// TIA Portal project "Automatic_Welder_1.0.0" (V19)
// Separate project file needed for simulation as  It was never possible to simulate an S7-1200 with firmware V3.0. It became only available with the firmware V4.0. Before this we had to use an S7-1500 to simulate the process.
// 
// The physical CPU cannot upgrade to firmware V3.0 -> V4.0. But software allows changing a V3.0 with V4.0 CPU. Downgrading a V4.0 project to V3.0 is not directly possible and is very painful.
// 
// The very best is to have two PLC projects. One is the design version (V3.0) and the other the simulation version (V4.0). Copy changes over from one to the other as needed.
// 
// The next option is to have a physical PLC at your desk. Ask your supplier to lend you a demo module from an old demo kit.

(* hardware
DEVICE "HMI_1"  TP700 Comfort
   slot 0: "HMI_1"  TP700 Comfort  6AV2 124-0GC01-0AX0  17.0.0.0
   slot 1: "HMI_1"  TP700 Comfort  6AV2 124-0GC01-0AX0  17.0.0.0
   slot 5: "HMI_1.IE_CP_1"  PROFINET Interface  17.0.0.0
      slot 1: "PROFINET Interface_1"  PROFINET Interface
         slot 1: "Port_1"  Port
         slot 2: "Port_2"  Port
   slot 7: "HMI_1.MPI/DP_CP_1"  MPI/DP Interface  17.0.0.0
DEVICE "S7-1200 station_1"  S7-1200 Station
   slot 0: "Rack_0"  S7-1200 Rack  Rack  V1.0
   slot 1: "PLC_1"  CPU 1214C DC/DC/DC  6ES7 214-1AG40-0XB0  V4.6
*)

// ===== PLC "PLC_1"  CPU 1214C DC/DC/DC =====

VAR_GLOBAL   // PLC tag table "Program Control"
   "ProgramStarted" AT %M0.1 : Bool;   // change to I instead of M later on
   "ProgramPaused" AT %M0.2 : Bool;   // change to I instead of M later on
   "SentCommandMoveXY" AT %M0.3 : Bool;   // being buggy and weird
   "SystemStatus" AT %QW1 : Int;   // codes: 100 - ok. 201 - motor address error
   "EnableMotorXY" AT %M0.0 : Bool;
END_VAR

VAR_GLOBAL   // PLC tag table "Clock_Memory"
   "Clock_Byte" AT %MB100 : Byte;
   "Clock_10Hz" AT %M100.0 : Bool;
   "Clock_5Hz" AT %M100.1 : Bool;
   "Clock_2.5Hz" AT %M100.2 : Bool;
   "Clock_2Hz" AT %M100.3 : Bool;
   "Clock_1.25Hz" AT %M100.4 : Bool;
   "Clock_1Hz" AT %M100.5 : Bool;
   "Clock_0.625Hz" AT %M100.6 : Bool;
   "Clock_0.5Hz" AT %M100.7 : Bool;
END_VAR

DATA_BLOCK "User_IO_DB"   // DB1
{ S7_Optimized_Access := 'TRUE' }
VERSION : 0.1
   VAR
      XSpeed : UDInt := 0;   // Pulse /hz
      XDest : UDInt;
      XPulses : DInt := 0;   // 21800 Pulse / 2mm
      XValue : UDInt := 0;   // 384-16=368u
      YSpeed : UDInt := 0;   // Pulse /hz
      YPulses : DInt := 0;   // 21800 Pulse / 2mm
      YDest : UDInt;
      Yvalue : UDInt := 0;   // 456-152=304u
   END_VAR
BEGIN
END_DATA_BLOCK

DATA_BLOCK "System_Update_DB"   // DB2
{ S7_Optimized_Access := 'TRUE' }
VERSION : 0.1
   VAR
      EnableMotorXYB : Bool;
      RunTerminationDone : Bool;
      RunStartupDone : Bool;
      DoneMotorX : Bool;
      DoneMotorXB : Bool;
      DoneMotorY : Bool;
      DoneMotorYB : Bool;
   END_VAR
BEGIN
END_DATA_BLOCK

DATA_BLOCK "Test_DB"   // DB3
{ S7_Optimized_Access := 'TRUE' }
VERSION : 0.1
   VAR
      "a" : DInt;
      aa : DInt;
      aaa : UDInt;
      aaaa : UDInt;
      "b" : Bool;
      bb : Bool;
      bbb : Bool;
      c : Time;
      dd : Real;
      d : Real;
      bbbb : Bool;
   END_VAR
BEGIN
END_DATA_BLOCK

// folder: Stepper Motor

DATA_BLOCK "X_Motor_Feedback_DB"   // DB5
{ S7_Optimized_Access := 'TRUE' }
VERSION : 0.1
// stored: InstanceOfName Motor_Feedback
"Motor_Feedback"
BEGIN
END_DATA_BLOCK

DATA_BLOCK "Y_Motor_Feedback_DB"   // DB6
{ S7_Optimized_Access := 'TRUE' }
VERSION : 0.1
// stored: InstanceOfName Motor_Feedback
"Motor_Feedback"
BEGIN
END_DATA_BLOCK

// folder: System blocks/Program resources

DATA_BLOCK "Motor_TimesUp_DB"   // DB4
{ S7_Optimized_Access := 'TRUE' }
AUTHOR : Simatic
FAMILY : IEC
NAME : IEC_TMR
VERSION : 1.0
// stored: InstanceOfName IEC_TIMER
"IEC_TIMER"
BEGIN
END_DATA_BLOCK

// folder: (top level)

ORGANIZATION_BLOCK "Main"   // OB1, LAD, ProgramCycle
TITLE = "Main Program Sweep (Cycle)"
{ S7_Optimized_Access := 'TRUE' }
VERSION : 0.1
   VAR_INPUT
      Initial_Call : Bool;   // Initial call of this OB
      Remanence : Bool;   // =True, if remanent data are available
   END_VAR
   VAR_TEMP
      XSucceeded : Bool;
      YSucceeded : Bool;
      Tmp : Bool;
      Tmp2 : Bool;
      TmpB : Bool;
   END_VAR
   VAR_TEMP   // added for the SCL form of the ladder/FBD networks
      _w1 : Bool;
      _w2 : Bool;
      _w3 : Bool;
      _w4 : Bool;
   END_VAR
BEGIN

REGION Network 1: Handle Motor UserInput
   // todo: need to size conversion for pulses, distance (mm), hmi distance (a.u.), del ismoving (redundant)
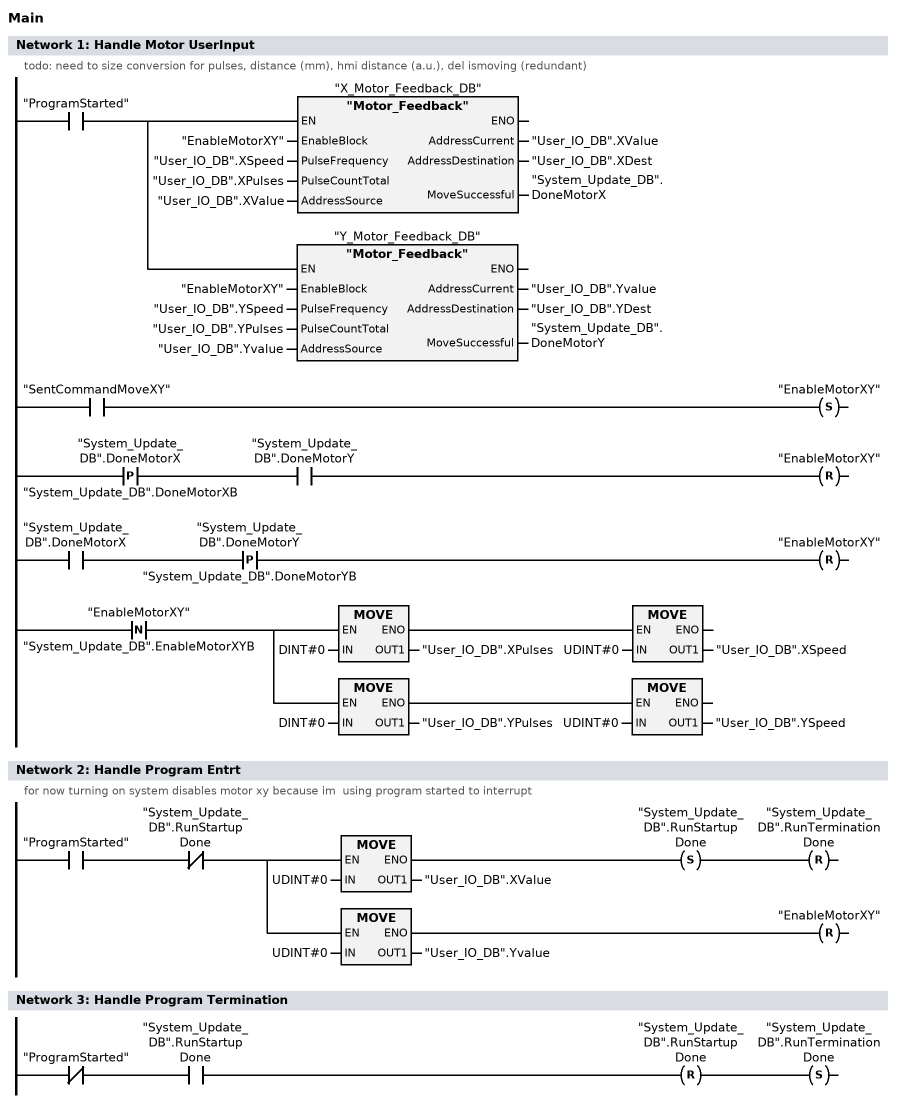
   RUNG wire#powerrail
      Contact( "ProgramStarted" )
      wire#w1
      "X_Motor_Feedback_DB"(EnableBlock := "EnableMotorXY", PulseFrequency := "User_IO_DB".XSpeed, PulseCountTotal := "User_IO_DB".XPulses, AddressSource := "User_IO_DB".XValue, AddressCurrent => "User_IO_DB".XValue, AddressDestination => "User_IO_DB".XDest, MoveSuccessful => "System_Update_DB".DoneMotorX)
   END_RUNG
   RUNG wire#w1
      "Y_Motor_Feedback_DB"(EnableBlock := "EnableMotorXY", PulseFrequency := "User_IO_DB".YSpeed, PulseCountTotal := "User_IO_DB".YPulses, AddressSource := "User_IO_DB".Yvalue, AddressCurrent => "User_IO_DB".Yvalue, AddressDestination => "User_IO_DB".YDest, MoveSuccessful => "System_Update_DB".DoneMotorY)
   END_RUNG
   RUNG wire#powerrail
      Contact( "SentCommandMoveXY" )
      S_Coil( "EnableMotorXY" )
   END_RUNG
   RUNG wire#powerrail
      P_Contact(operand := "System_Update_DB".DoneMotorX, bit := "System_Update_DB".DoneMotorXB)
      Contact( "System_Update_DB".DoneMotorY )
      R_Coil( "EnableMotorXY" )
   END_RUNG
   RUNG wire#powerrail
      Contact( "System_Update_DB".DoneMotorX )
      P_Contact(operand := "System_Update_DB".DoneMotorY, bit := "System_Update_DB".DoneMotorYB)
      R_Coil( "EnableMotorXY" )
   END_RUNG
   RUNG wire#powerrail
      N_Contact(operand := "EnableMotorXY", bit := "System_Update_DB".EnableMotorXYB)
      wire#w2
      Move(in := DINT#0, out1 => "User_IO_DB".XPulses)
      Move(in := UDINT#0, out1 => "User_IO_DB".XSpeed)
   END_RUNG
   RUNG wire#w2
      Move(in := DINT#0, out1 => "User_IO_DB".YPulses)
      Move(in := UDINT#0, out1 => "User_IO_DB".YSpeed)
   END_RUNG
   // the same network as SCL:
   #_w1 := "ProgramStarted";
   IF #_w1 THEN
       "X_Motor_Feedback_DB"(EnableBlock := "EnableMotorXY",   // "Motor_Feedback"
                             PulseFrequency := "User_IO_DB".XSpeed,
                             PulseCountTotal := "User_IO_DB".XPulses,
                             AddressSource := "User_IO_DB".XValue,
                             AddressCurrent => "User_IO_DB".XValue,
                             AddressDestination => "User_IO_DB".XDest,
                             MoveSuccessful => "System_Update_DB".DoneMotorX);
       "Y_Motor_Feedback_DB"(EnableBlock := "EnableMotorXY",   // "Motor_Feedback"
                             PulseFrequency := "User_IO_DB".YSpeed,
                             PulseCountTotal := "User_IO_DB".YPulses,
                             AddressSource := "User_IO_DB".Yvalue,
                             AddressCurrent => "User_IO_DB".Yvalue,
                             AddressDestination => "User_IO_DB".YDest,
                             MoveSuccessful => "System_Update_DB".DoneMotorY);
   END_IF;
   IF "SentCommandMoveXY" THEN "EnableMotorXY" := TRUE; END_IF;
   #_w2 := "System_Update_DB".DoneMotorX AND NOT "System_Update_DB".DoneMotorXB;   // rising edge of "System_Update_DB".DoneMotorX
   "System_Update_DB".DoneMotorXB := "System_Update_DB".DoneMotorX;
   IF #_w2 AND "System_Update_DB".DoneMotorY THEN "EnableMotorXY" := FALSE; END_IF;
   #_w3 := "System_Update_DB".DoneMotorX AND "System_Update_DB".DoneMotorY AND NOT "System_Update_DB".DoneMotorYB;   // rising edge of "System_Update_DB".DoneMotorY
   "System_Update_DB".DoneMotorYB := "System_Update_DB".DoneMotorY;
   IF #_w3 THEN "EnableMotorXY" := FALSE; END_IF;
   #_w4 := NOT "EnableMotorXY" AND "System_Update_DB".EnableMotorXYB;   // falling edge of "EnableMotorXY"
   "System_Update_DB".EnableMotorXYB := "EnableMotorXY";
   IF #_w4 THEN
       "User_IO_DB".XPulses := DINT#0;
       "User_IO_DB".XSpeed := UDINT#0;
       "User_IO_DB".YPulses := DINT#0;
       "User_IO_DB".YSpeed := UDINT#0;
   END_IF;
END_REGION

REGION Network 2: Handle Program Entrt
   // for now turning on system disables motor xy because im  using program started to interrupt
   RUNG wire#powerrail
      Contact( "ProgramStarted" )
      I_Contact( "System_Update_DB".RunStartupDone )
      wire#w1
      Move(in := UDINT#0, out1 => "User_IO_DB".XValue)
      S_Coil( "System_Update_DB".RunStartupDone )
      R_Coil( "System_Update_DB".RunTerminationDone )
   END_RUNG
   RUNG wire#w1
      Move(in := UDINT#0, out1 => "User_IO_DB".Yvalue)
      R_Coil( "EnableMotorXY" )
   END_RUNG
   // the same network as SCL:
   IF "ProgramStarted" AND NOT "System_Update_DB".RunStartupDone THEN "User_IO_DB".XValue := UDINT#0; END_IF;
   #_w1 := "ProgramStarted" AND NOT "System_Update_DB".RunStartupDone;
   IF #_w1 THEN
       "System_Update_DB".RunStartupDone := TRUE;
       "System_Update_DB".RunTerminationDone := FALSE;
       "User_IO_DB".Yvalue := UDINT#0;
       "EnableMotorXY" := FALSE;
   END_IF;
END_REGION

REGION Network 3: Handle Program Termination
   RUNG wire#powerrail
      I_Contact( "ProgramStarted" )
      Contact( "System_Update_DB".RunStartupDone )
      R_Coil( "System_Update_DB".RunStartupDone )
      S_Coil( "System_Update_DB".RunTerminationDone )
   END_RUNG
   // the same network as SCL:
   #_w1 := NOT "ProgramStarted" AND "System_Update_DB".RunStartupDone;
   IF #_w1 THEN
       "System_Update_DB".RunStartupDone := FALSE;
       "System_Update_DB".RunTerminationDone := TRUE;
   END_IF;
END_REGION
END_ORGANIZATION_BLOCK

ORGANIZATION_BLOCK "Test_CyclicOB"   // OB123, LAD, ProgramCycle
TITLE = "Main Program Sweep (Cycle)"
{ S7_Optimized_Access := 'TRUE' }
VERSION : 0.1
   VAR_INPUT
      Initial_Call : Bool;   // Initial call of this OB
      Remanence : Bool;   // =True, if remanent data are available
   END_VAR
   VAR_TEMP
      tb : Bool;
      tbb : Bool;
      var_time1 : Real;
      var_time2 : UDInt;
      tbEdgeDetected : Bool;
   END_VAR
   VAR_TEMP   // added for the SCL form of the ladder/FBD networks
      _w1 : Bool;
   END_VAR
BEGIN

REGION Network 1: Ladder logic (I am retarded)
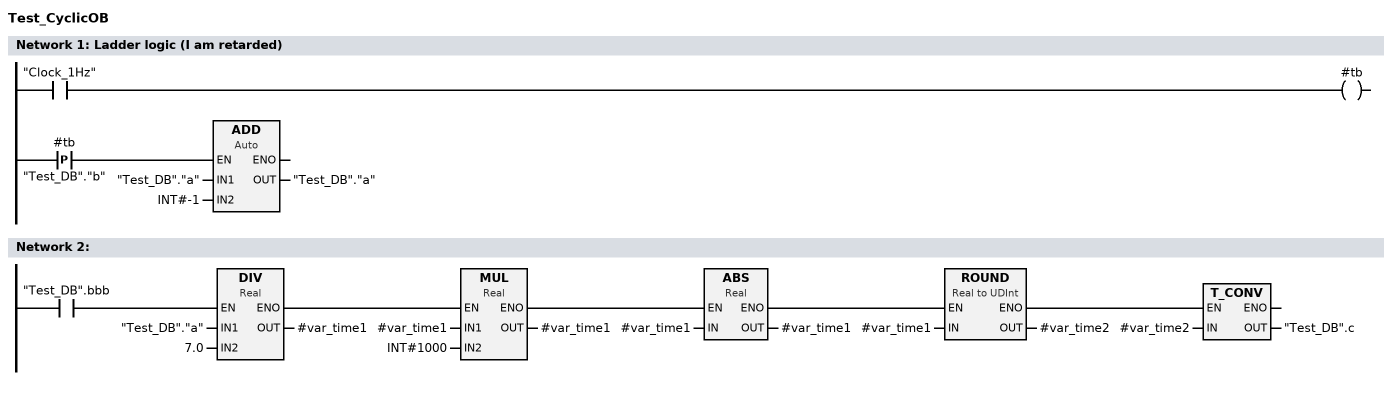
   RUNG wire#powerrail
      Contact( "Clock_1Hz" )
      Coil( #tb )
   END_RUNG
   RUNG wire#powerrail
      P_Contact(operand := #tb, bit := "Test_DB"."b")
      Add(in1 := "Test_DB"."a", in2 := INT#-1, out => "Test_DB"."a")
   END_RUNG
   // the same network as SCL:
   #tb := "Clock_1Hz";
   #_w1 := #tb AND NOT "Test_DB"."b";   // rising edge of #tb
   "Test_DB"."b" := #tb;
   IF #_w1 THEN "Test_DB"."a" := "Test_DB"."a" + INT#-1; END_IF;
END_REGION

REGION Network 2
   IF "Test_DB".bbb THEN
       #var_time1 := "Test_DB"."a" / 7.0;
       #var_time1 := #var_time1 * INT#1000;
       #var_time1 := ABS(#var_time1);
       #var_time2 := ROUND(#var_time1);
       "Test_DB".c := T_CONV(IN := #var_time2);
   END_IF;
END_REGION

REGION Network 3 (SCL): turn pulses into time (ms)
   #var_time1 := "Test_DB".a / 7;
   #var_time1 := ABS(#var_time1 * 1000);
   #var_time2 := REAL_TO_UDINT(#var_time1);
   "Test_DB".c := UDINT_TO_TIME(#var_time2);
END_REGION
END_ORGANIZATION_BLOCK

// folder: Stepper Motor

FUNCTION_BLOCK "Motor_Feedback"   // FB2, LAD
TITLE = Motor Telemetry: Get current axis position and if the motor is moving.
{ S7_Optimized_Access := 'TRUE' }
VERSION : 0.1
// TODO: Make block figure out when to allow the motor to stop moving (So that the current location is known.) when a move operation is interrupted.
// Implement reversed movement logic
// 
// Motor movement logic is currently only in blocks of pulse per 500ms except for final, ratify this.
// go test if can change the static vars to temp
// 
// d = vt
// pulses = pulsefrequency times time
// go figure out how far one pulse moves,  bi/unipolar, do conversions to metric!
   VAR_INPUT
      EnableBlock : Bool;
      PulseFrequency : DInt;   // hz
      PulseCountTotal : DInt;
      AddressSource : DInt;
   END_VAR
   VAR_OUTPUT
      AddressCurrent : DInt;
      AddressDestination : Int;
      MoveSuccessful : Bool;
   END_VAR
   VAR
      TimeTotalms : Time;
      PulseCountDone : DInt;
      Movement500ms : DInt;
      IsMoving : Bool;
      IsMovingM : Bool;
      TimerDiff : Bool;
      TimerDiffB : Bool;
      EnableBlockM : Bool;
   END_VAR
   VAR_TEMP
      IsPulseCountNegative : SInt;
      PulseCountAbs : UDInt;
   END_VAR
   VAR_TEMP   // added for the SCL form of the ladder/FBD networks
      _w1 : Bool;
      _w2 : Bool;
   END_VAR
BEGIN

REGION Network 1: ENTRY Evaluate Working Variables + Call Main
   // I spent 2 hours on this: Scan Op for positve edge can only be used for one row! This is because it ref the same bit.
   // 
   // Find:
   // - Move Destination
   // - Time total (ms): PulseCountTotal = PulseFrequency(hz) * Time (s)
   // - Pulses / 500ms (auto rounded by DIV)
   // - Current Address = Source Address
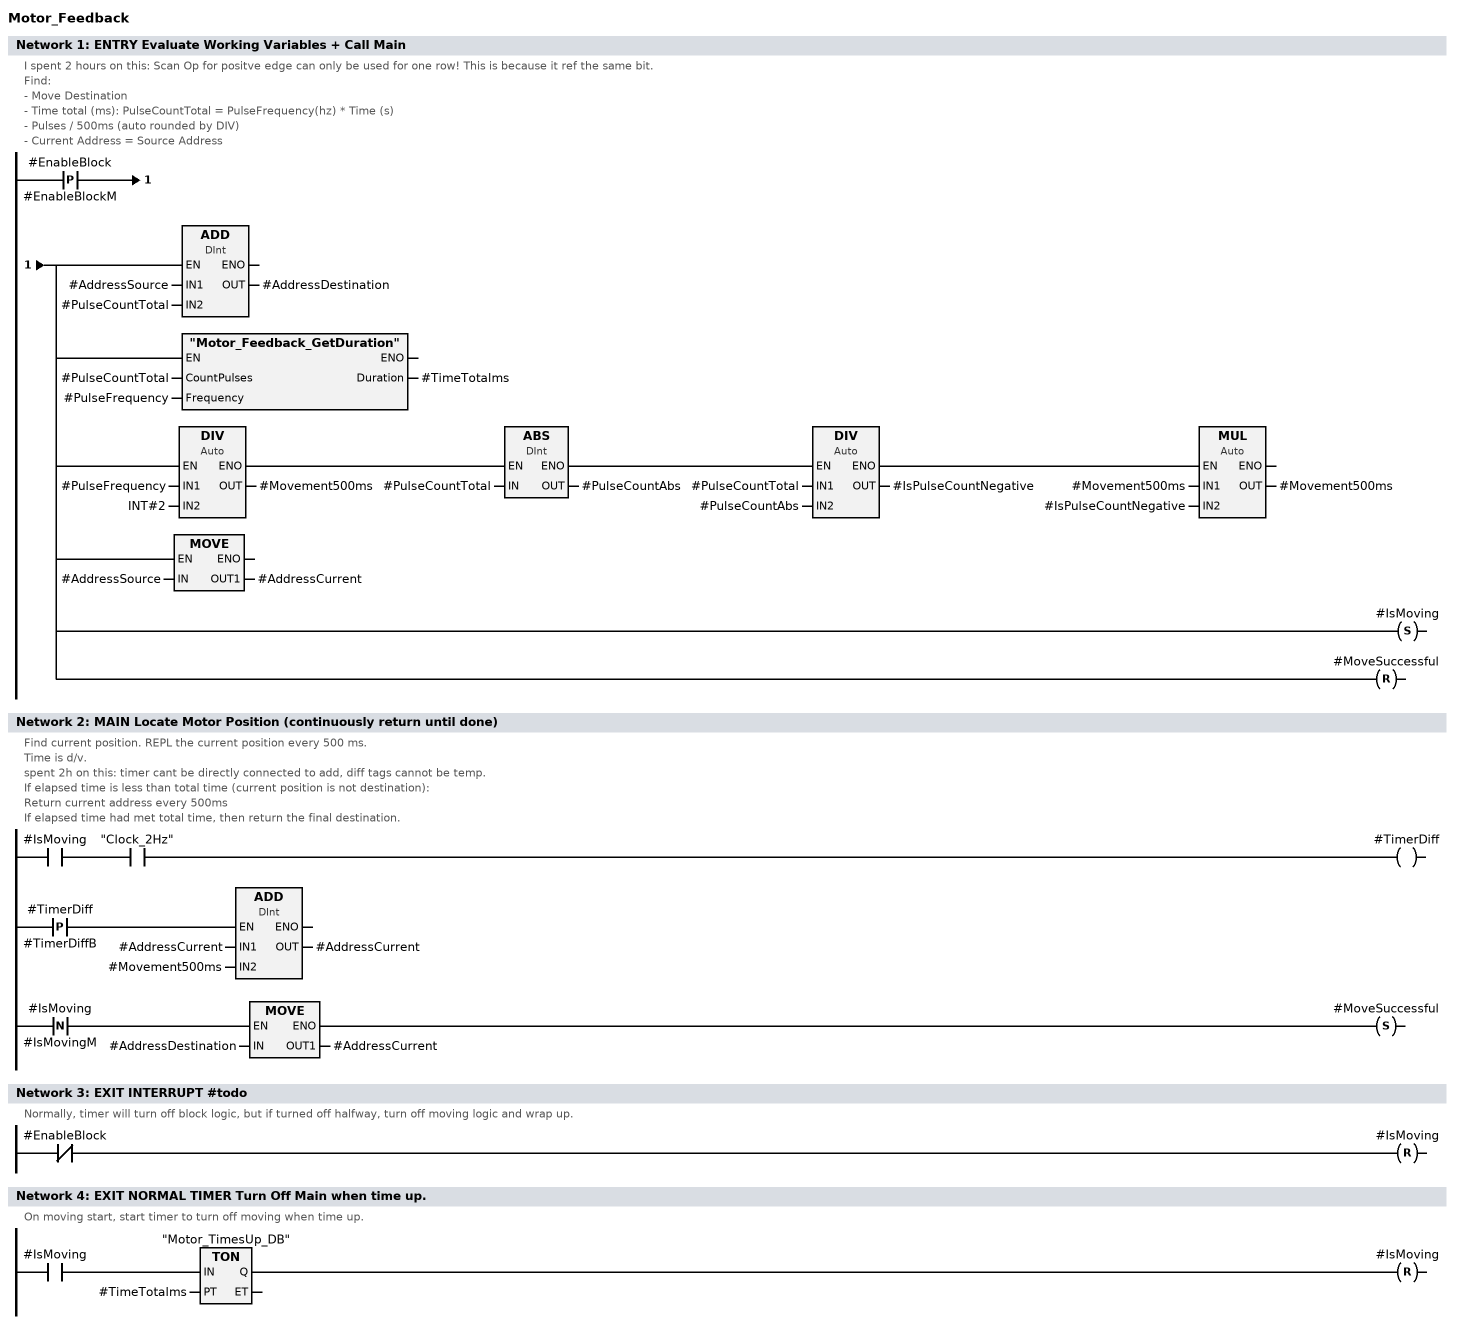
   RUNG wire#powerrail
      P_Contact(operand := #EnableBlock, bit := #EnableBlockM)
      wire#w1
      { S7_Templates := "SrcType := DInt" } Add(in1 := #AddressSource, in2 := #PulseCountTotal, out => #AddressDestination)
   END_RUNG
   RUNG wire#w1
      "Motor_Feedback_GetDuration"(CountPulses := #PulseCountTotal, Frequency := #PulseFrequency, Duration => #TimeTotalms)
   END_RUNG
   RUNG wire#w1
      Div(in1 := #PulseFrequency, in2 := INT#2, out => #Movement500ms)
      { S7_Templates := "SrcType := DInt" } Abs(in := #PulseCountTotal, out => #PulseCountAbs)
      Div(in1 := #PulseCountTotal, in2 := #PulseCountAbs, out => #IsPulseCountNegative)
      Mul(in1 := #Movement500ms, in2 := #IsPulseCountNegative, out => #Movement500ms)
   END_RUNG
   RUNG wire#w1
      Move(in := #AddressSource, out1 => #AddressCurrent)
   END_RUNG
   RUNG wire#w1
      S_Coil( #IsMoving )
   END_RUNG
   RUNG wire#w1
      R_Coil( #MoveSuccessful )
   END_RUNG
   // the same network as SCL:
   #_w1 := #EnableBlock AND NOT #EnableBlockM;   // rising edge of #EnableBlock
   #EnableBlockM := #EnableBlock;
   IF #_w1 THEN
       #AddressDestination := #AddressSource + #PulseCountTotal;
       "Motor_Feedback_GetDuration"(CountPulses := #PulseCountTotal,
                               Frequency := #PulseFrequency,
                               Duration => #TimeTotalms);
       #Movement500ms := #PulseFrequency / INT#2;
       #PulseCountAbs := ABS(#PulseCountTotal);
       #IsPulseCountNegative := #PulseCountTotal / #PulseCountAbs;
       #Movement500ms := #Movement500ms * #IsPulseCountNegative;
       #AddressCurrent := #AddressSource;
       #IsMoving := TRUE;
       #MoveSuccessful := FALSE;
   END_IF;
END_REGION

REGION Network 2: MAIN Locate Motor Position (continuously return until done)
   // Find current position. REPL the current position every 500 ms.
   // Time is d/v. 
   // 
   // spent 2h on this: timer cant be directly connected to add, diff tags cannot be temp.
   // 
   // If elapsed time is less than total time (current position is not destination):
   // Return current address every 500ms
   // 
   // If elapsed time had met total time, then return the final destination.
   RUNG wire#powerrail
      Contact( #IsMoving )
      Contact( "Clock_2Hz" )
      Coil( #TimerDiff )
   END_RUNG
   RUNG wire#powerrail
      P_Contact(operand := #TimerDiff, bit := #TimerDiffB)
      { S7_Templates := "SrcType := DInt" } Add(in1 := #AddressCurrent, in2 := #Movement500ms, out => #AddressCurrent)
   END_RUNG
   RUNG wire#powerrail
      N_Contact(operand := #IsMoving, bit := #IsMovingM)
      Move(in := #AddressDestination, out1 => #AddressCurrent)
      S_Coil( #MoveSuccessful )
   END_RUNG
   // the same network as SCL:
   #TimerDiff := #IsMoving AND "Clock_2Hz";
   #_w1 := #TimerDiff AND NOT #TimerDiffB;   // rising edge of #TimerDiff
   #TimerDiffB := #TimerDiff;
   IF #_w1 THEN #AddressCurrent := #AddressCurrent + #Movement500ms; END_IF;
   #_w2 := NOT #IsMoving AND #IsMovingM;   // falling edge of #IsMoving
   #IsMovingM := #IsMoving;
   IF #_w2 THEN
       #AddressCurrent := #AddressDestination;
       #MoveSuccessful := TRUE;
   END_IF;
END_REGION

REGION Network 3: EXIT INTERRUPT #todo
   // Normally, timer will turn off block logic, but if turned off halfway, turn off moving logic and wrap up.
   RUNG wire#powerrail
      I_Contact( #EnableBlock )
      R_Coil( #IsMoving )
   END_RUNG
   // the same network as SCL:
   IF NOT #EnableBlock THEN #IsMoving := FALSE; END_IF;
END_REGION

REGION Network 4: EXIT NORMAL TIMER Turn Off Main when time up.
   // On moving start, start timer to turn off moving when time up.
   "Motor_TimesUp_DB".TON(IN := #IsMoving, PT := #TimeTotalms);
   IF "Motor_TimesUp_DB".Q THEN #IsMoving := FALSE; END_IF;
END_REGION
END_FUNCTION_BLOCK

FUNCTION_BLOCK "Motor_Commands"   // FB3, LAD
{ S7_Optimized_Access := 'TRUE' }
VERSION : 0.1
   VAR_OUTPUT
      Pulse : Bool;
   END_VAR
BEGIN
END_FUNCTION_BLOCK

FUNCTION "Motor_Feedback_GetDuration" : Void   // FC1, SCL
{ S7_Optimized_Access := 'TRUE' }
VERSION : 0.1
   VAR_INPUT
      CountPulses : DInt;
      Frequency : DInt;
   END_VAR
   VAR_OUTPUT
      Duration : Time;
   END_VAR
   VAR_TEMP
      x0 : Real;
      x1 : UDInt;
   END_VAR
BEGIN
   #x0 := #CountPulses / #Frequency; // real output
   #x0 := ABS(#x0 * 1000);
   #x1 := REAL_TO_UDINT(#x0);
   #Duration := UDINT_TO_TIME(#x1);
END_FUNCTION

FUNCTION "Motor_Feedback_GetMovement" : Void   // FC2, LAD
{ S7_Optimized_Access := 'TRUE' }
VERSION : 0.1
   VAR_INPUT
      PulseFrequency : UDInt;
      PulseCount : DInt;
      ClockInterval : USInt;
   END_VAR
   VAR_OUTPUT
      MovementUnit : DInt;
   END_VAR
   VAR_TEMP
      PulseCountAbs : UDInt;
      IsPulseCountNegative : SInt;
      MovementUnitAbs : UDInt;
   END_VAR
BEGIN

REGION Network 1
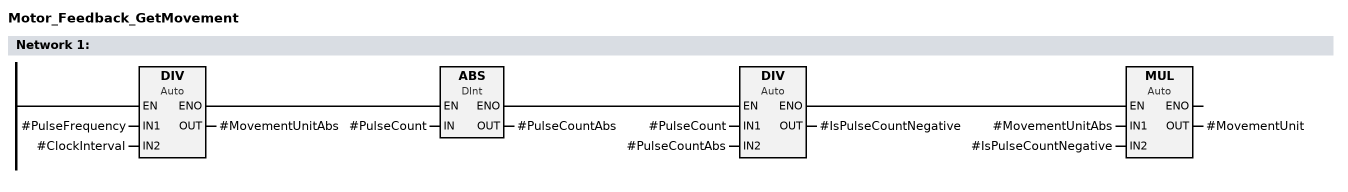
   RUNG wire#powerrail
      Div(in1 := #PulseFrequency, in2 := #ClockInterval, out => #MovementUnitAbs)
      { S7_Templates := "SrcType := DInt" } Abs(in := #PulseCount, out => #PulseCountAbs)
      Div(in1 := #PulseCount, in2 := #PulseCountAbs, out => #IsPulseCountNegative)
      Mul(in1 := #MovementUnitAbs, in2 := #IsPulseCountNegative, out => #MovementUnit)
   END_RUNG
   // the same network as SCL:
   #MovementUnitAbs := #PulseFrequency / #ClockInterval;
   #PulseCountAbs := ABS(#PulseCount);
   #IsPulseCountNegative := #PulseCount / #PulseCountAbs;
   #MovementUnit := #MovementUnitAbs * #IsPulseCountNegative;
END_REGION
END_FUNCTION

(* ===== HMI "HMI_1" =====
system functions are stored by id; their names below are inferred from use
connection "HMI_Connection_2": ETHERNET, S7_1200_OMS

HMI tags "Default tag table"
   "ProgramStarted" : Bool = PLC ProgramStarted AT %M0.1, 1 s
   "SentCommandMoveXY" : Bool = PLC SentCommandMoveXY AT %M0.3, 1 s
   "XValue" : UDInt = PLC User_IO_DB.XValue AT %ID18, 1 s
   "YValue" : UDInt = PLC User_IO_DB.Yvalue AT %ID22, 1 s
   "Error" : Int, internal
   "User_Input_DB_XSpeed" : UDInt = PLC User_IO_DB.XSpeed, 1 s
   "User_Input_DB_XPulses" : DInt = PLC User_IO_DB.XPulses, 1 s
   "User_Input_DB_YSpeed" : UDInt = PLC User_IO_DB.YSpeed, 1 s
   "User_Input_DB_YPulses" : DInt = PLC User_IO_DB.YPulses, 1 s
   "ProgramPaused" : Bool = PLC ProgramPaused AT %M0.2, 1 s
   "Test_DB_a" : DInt = PLC Test_DB.a, 1 s

HMI tags "HMI Only (Not Powertags)"
   "sussy amogus" : Int, internal

recipe "2 Axis Movements": X Pulses <- "User_Input_DB_XPulses", X Speed <- "User_Input_DB_XSpeed", Y Pulses <- "User_Input_DB_YPulses", Y Speed <- "User_Input_DB_YSpeed"

screen "Map + Recipe" 800x479
   Rectangle "graph bg" at 16,120 size 376x312
      Appearance <- "Error"
   Circle "Weld" at 16,120 size 8x8
      DirectMovement <- "XValue"
      DirectMovement <- "YValue"
   Button "Page" at 296,440 size 96x32; TextOff 'Next pg'
      on Click: ActivateScreen("Testing screen", 0)
   Switch "program start" at 16,440 size 96x32; CaptionText 'Switch'; TextOff 'OFF'; TextOn 'ON'
      on SwitchOn: SetBit("ProgramStarted")
      on SwitchOff: ResetBit("ProgramStarted")
      ProcessValue <- "ProgramStarted"
   Button "program pause" at 152,440 size 96x32; TextOff 'Pause'
      Appearance <- "ProgramPaused"
      on Release: InvertBit("ProgramPaused")
   IOField "y pulses" at 104,72 size 48x32; FormatPattern 999
      ProcessValue <- "YValue"
   IOField "x speed" at 48,40 size 56x32; FormatPattern 9999
      ProcessValue <- "User_Input_DB_XSpeed"
   IOField "y speed" at 48,72 size 56x32; FormatPattern 9999
      ProcessValue <- "User_Input_DB_YSpeed"
   IOField "x pulses" at 104,40 size 48x32; FormatPattern 999
      ProcessValue <- "XValue"
   TextField "speed" at 48,16 size 60x23; Text 'Speed'
   TextField "x" at 24,40 size 17x23; Text 'X'
   TextField "y" at 24,72 size 17x23; Text 'Y'
   TextField "pulses" at 104,16 size 56x23; Text 'Value'
   Button "send move command" at 296,56 size 96x32; TextOff 'Send'
      Appearance <- "SentCommandMoveXY"
      on Press: function_b14e0dd5("SentCommandMoveXY", 0)
   RecipeView "Recipe view_1" at 408,0 size 392x474
   Circle "Weld_Guide" at 16,120 size 8x8
      DirectMovement <- "XValue"
      DirectMovement <- "YValue"

screen "Testing screen" 800x479
   IOField "I/O field_1" at 40,64 size 96x32; FormatPattern 9999999999
      ProcessValue <- "XValue"
   IOField "I/O field_3" at 40,96 size 96x32; FormatPattern s9999999999
      ProcessValue <- "User_Input_DB_XPulses"
   Button "Button_1" at 40,160 size 96x32; TextOff 'next pg'
      on Click: ActivateScreen("Map + Recipe", 0)
   IOField "I/O field_4" at 40,128 size 96x32; FormatPattern s9999999999
      ProcessValue <- "Test_DB_a"
   StatusForce "Watch table_1" at 200,0 size 600x444; ToolTipText 'Text'
*)